// TIA Portal V19 export
TYPE "Positioning_EPOS_Machine_Manager"
// stored: Access Published
   STRUCT
      EnableStopDoorOpeningReq : Bool;
      EnableStopInPhase : Bool;
      EnableStopProgrammed : Bool;
      Control_ON : Bool;
      Minus : Bool;   // Move in negative direction
      Plus : Bool;   // Move in positive direction
      MoveToPos : Bool;   // Move to target position
      Pos : LReal;   // [mm] Target position
      Vel : LReal;   // [mm/min]
      Acc : LReal;   // [mm/s²]
      Dec : LReal;   // [mm/s²]
   END_STRUCT;
END_TYPE
